// LS Electric XG5000 project: Test_unity
// PLC LSPLC

PROGRAM NewProgram (task: 스캔 프로그램)

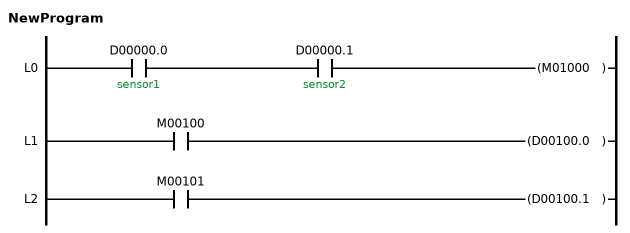
; L0
LOAD      D00000.0	// sensor1
AND       D00000.1	// sensor2
OUT       M01000
; L1
LOAD      M00100
OUT       D00100.0
; L2
LOAD      M00101
OUT       D00100.1